(* PLC project Rasi_feeds_batching2.project, Automation Builder 2.7 - Basic Automation Builder 2.7 *)
(* stored: creationDateTime 2026-09-03T18:55:00.218576, modificationDateTime 2026-09-01T07:53:31.7371227 *)

PROGRAM batching14
  VAR
    Auto_Ctrl : Auto_Batching_V14;
    Semi_Auto_Ctrl : Semi_Auto_Batching_V14;
    Auto_Complete : BOOL;
    Semi_Auto_Complete : BOOL;
    Auto_Err : INT;
    Auto_Msg : STRING;
    Semi_Auto_Err : INT;
    Semi_Auto_Msg : STRING;
    FB_Samyak_Multi_1 : FB_Samyak_Multi;
    arrSlaveIDs : ARRAY[1..4] OF BYTE := [1, 2, 0, 0];
    arrDivisor : ARRAY[1..4] OF REAL := [10.0, 10.0, 1.0, 1.0];
    arrTare_In : ARRAY[1..4] OF BOOL;
    Weight_Scaled_Array : ARRAY[1..4] OF REAL;
    arrLine_Fault : ARRAY[1..4] OF BOOL;
  END_VAR

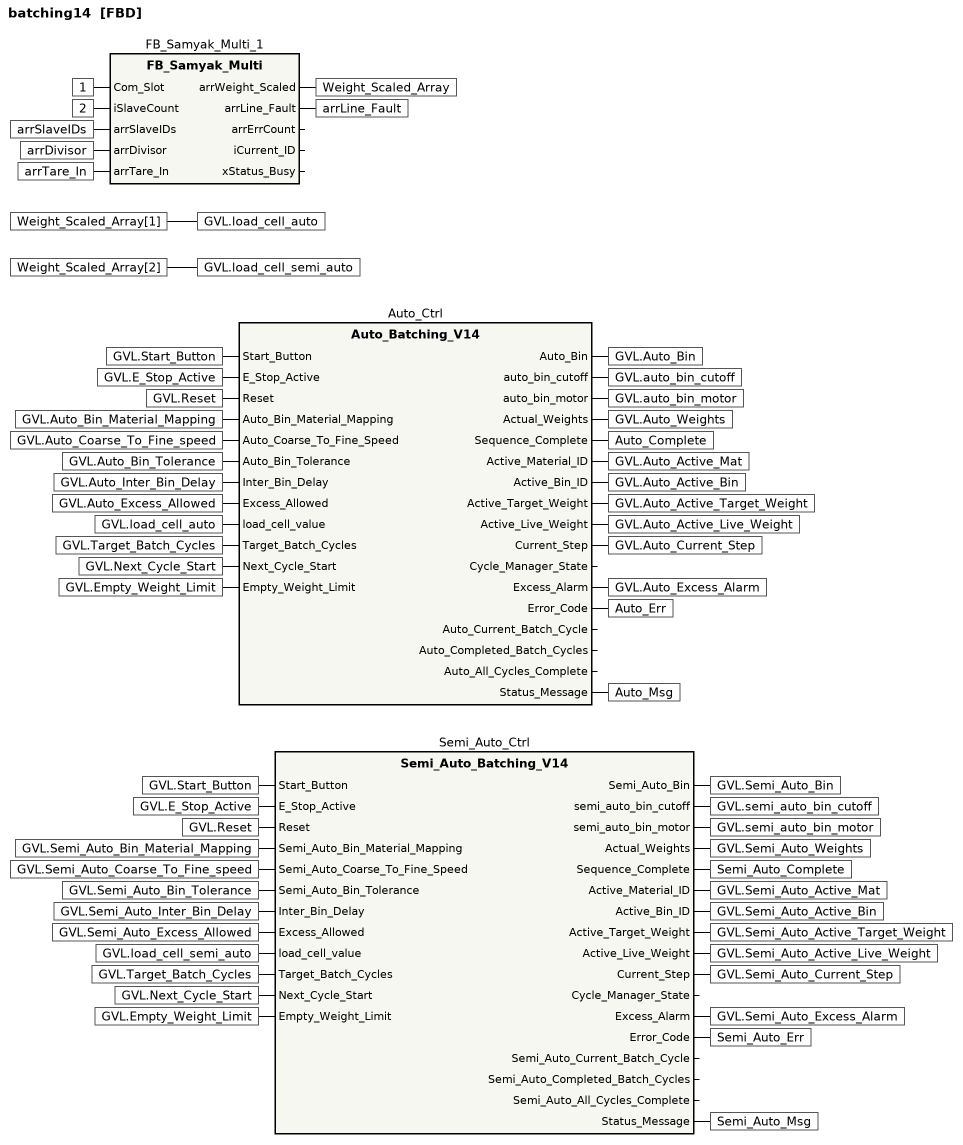
(* FBD diagram, written out as Structured Text *)
FB_Samyak_Multi_1(Com_Slot := 1, iSlaveCount := 2, arrSlaveIDs := arrSlaveIDs, arrDivisor := arrDivisor, arrTare_In := arrTare_In, arrLine_Fault => arrLine_Fault);
Weight_Scaled_Array := FB_Samyak_Multi_1.arrWeight_Scaled;
GVL.load_cell_auto := Weight_Scaled_Array[1];
GVL.load_cell_semi_auto := Weight_Scaled_Array[2];
Auto_Ctrl(Start_Button := GVL.Start_Button, E_Stop_Active := GVL.E_Stop_Active, Reset := GVL.Reset, Auto_Bin_Material_Mapping := GVL.Auto_Bin_Material_Mapping, Auto_Coarse_To_Fine_Speed := GVL.Auto_Coarse_To_Fine_speed, Auto_Bin_Tolerance := GVL.Auto_Bin_Tolerance, Inter_Bin_Delay := GVL.Auto_Inter_Bin_Delay, Excess_Allowed := GVL.Auto_Excess_Allowed, load_cell_value := GVL.load_cell_auto, Target_Batch_Cycles := GVL.Target_Batch_Cycles, Next_Cycle_Start := GVL.Next_Cycle_Start, Empty_Weight_Limit := GVL.Empty_Weight_Limit, auto_bin_cutoff => GVL.auto_bin_cutoff, auto_bin_motor => GVL.auto_bin_motor, Actual_Weights => GVL.Auto_Weights, Sequence_Complete => Auto_Complete, Active_Material_ID => GVL.Auto_Active_Mat, Active_Bin_ID => GVL.Auto_Active_Bin, Active_Target_Weight => GVL.Auto_Active_Target_Weight, Active_Live_Weight => GVL.Auto_Active_Live_Weight, Current_Step => GVL.Auto_Current_Step, Excess_Alarm => GVL.Auto_Excess_Alarm, Error_Code => Auto_Err, Status_Message => Auto_Msg);
GVL.Auto_Bin := Auto_Ctrl.Auto_Bin;
Semi_Auto_Ctrl(Start_Button := GVL.Start_Button, E_Stop_Active := GVL.E_Stop_Active, Reset := GVL.Reset, Semi_Auto_Bin_Material_Mapping := GVL.Semi_Auto_Bin_Material_Mapping, Semi_Auto_Coarse_To_Fine_Speed := GVL.Semi_Auto_Coarse_To_Fine_speed, Semi_Auto_Bin_Tolerance := GVL.Semi_Auto_Bin_Tolerance, Inter_Bin_Delay := GVL.Semi_Auto_Inter_Bin_Delay, Excess_Allowed := GVL.Semi_Auto_Excess_Allowed, load_cell_value := GVL.load_cell_semi_auto, Target_Batch_Cycles := GVL.Target_Batch_Cycles, Next_Cycle_Start := GVL.Next_Cycle_Start, Empty_Weight_Limit := GVL.Empty_Weight_Limit, semi_auto_bin_cutoff => GVL.semi_auto_bin_cutoff, semi_auto_bin_motor => GVL.semi_auto_bin_motor, Actual_Weights => GVL.Semi_Auto_Weights, Sequence_Complete => Semi_Auto_Complete, Active_Material_ID => GVL.Semi_Auto_Active_Mat, Active_Bin_ID => GVL.Semi_Auto_Active_Bin, Active_Target_Weight => GVL.Semi_Auto_Active_Target_Weight, Active_Live_Weight => GVL.Semi_Auto_Active_Live_Weight, Current_Step => GVL.Semi_Auto_Current_Step, Excess_Alarm => GVL.Semi_Auto_Excess_Alarm, Error_Code => Semi_Auto_Err, Status_Message => Semi_Auto_Msg);
GVL.Semi_Auto_Bin := Semi_Auto_Ctrl.Semi_Auto_Bin;
END_PROGRAM
